FUNCTION_BLOCK FB_MyBlock
VAR_OUTPUT
	myVar		: INT := 42;
END_VAR

END_FUNCTION_BLOCK

(* stored: Version 1.1.0.1
   POU FB_MyBlock: Id {f43557f1-a608-470a-a7b8-6c4150ab7563}, SpecialFunc None *)
